PROGRAM SafetyInterface_Enc053
VAR
	{attribute 'TcLinkTo' := '
		.iSafteyCtrlProjectCRC := TIIB[N20S14 (EL6910)]^Device Info Data^Project CRC;
		.iSafetyGroup_State := TIIB[N20S14 (EL6910)]^TwinSAFE Group Info Data^Enc053_SafetyGroup Info Data^State;
		.iSafetyGroup_Diag := TIIB[N20S14 (EL6910)]^TwinSAFE Group Info Data^Enc053_SafetyGroup Info Data^Diag;
		.iSafetyGroup_ComErr := TIIB[N20S14 (EL6910)]^StandardInputs^Enc053_SafetyGroup.oGroup_ComErr_3;
		.iSafetyGroup_ComInStartup := TIIB[N20S14 (EL6910)]^StandardInputs^Enc053_SafetyGroup.oGroup_ComInStartup_4;
		.iSafetyGroup_FBErr := TIIB[N20S14 (EL6910)]^StandardInputs^Enc053_SafetyGroup.oGroup_FBErr_5;
		.iSafetyGroup_FBInRun := TIIB[N20S14 (EL6910)]^StandardInputs^Enc053_SafetyGroup.oGroup_FBInRun_6;
		.iSafetyGroup_InRun := TIIB[N20S14 (EL6910)]^StandardInputs^Enc053_SafetyGroup.oGroup_InRun_7;
		.iSafetyGroup_OtherErr := TIIB[N20S14 (EL6910)]^StandardInputs^Enc053_SafetyGroup.oGroup_OtherErr_8;
		.oSafetyGroup_ErrAck := TIIB[N20S14 (EL6910)]^StandardOutputs^Enc053_SafetyGroup.iGroup_ErrAck_1;
		.oSafetyGroup_Run := TIIB[N20S14 (EL6910)]^StandardOutputs^Enc053_SafetyGroup.iGroup_Run_2;
		.oControlPowerPBLight := TIIB[N20S09 (EL2008)]^Channel 1^Output;
		.iSafetyResetPB := TIIB[N20S14 (EL6910)]^Connection Info Data^Enc053_SafetyGroup.N20S01 Digital 4 In (EL1904)_9 Info Data^Input Safe Data InputChannel3;
		.iEstopPB1_CH1 := TIIB[N20S14 (EL6910)]^Connection Info Data^Enc053_SafetyGroup.N20S01 Digital 4 In (EL1904)_9 Info Data^Input Safe Data InputChannel1;
		.iEstopPB1_CH2 := TIIB[N20S14 (EL6910)]^Connection Info Data^Enc053_SafetyGroup.N20S01 Digital 4 In (EL1904)_9 Info Data^Input Safe Data InputChannel2;
		.iRelayNCContact_Estop := TIIB[N20S14 (EL6910)]^Connection Info Data^Enc053_SafetyGroup.N20S03 Digital 4 In (EL1904)_11 Info Data^Input Safe Data InputChannel1;
		.iSafetyPowerOn_Estop_CH1 := TIIB[N20S14 (EL6910)]^Connection Info Data^Enc053_SafetyGroup.N20S04 Digital 4 Out (EL2904)_20 Info Data^Output Safe Data OutputChannel1;
		.iSafetyPowerOn_Estop_CH2 := TIIB[N20S14 (EL6910)]^Connection Info Data^Enc053_SafetyGroup.N20S04 Digital 4 Out (EL2904)_20 Info Data^Output Safe Data OutputChannel2;
		.iAirPressureOk := TIIB[N20S06 (EL1008)]^Channel 2^Input'}
	fbSafetyInterface : FB_SafetyInterfaceConv;
END_VAR



fbSafetyInterface(
	pSafetyInterface := ADR(gProduced_SafetyInterfaceConv.Enc053));

END_PROGRAM

(* stored: Version 1.1.0.1, ProductVersion 3.1.4024.6
   POU SafetyInterface_Enc053: Id {3e8fa51f-9045-4f3f-beb2-7d76f8764eae}, SpecialFunc None *)
